TYPE DMC_Ins :
STRUCT
	DMC_Inputs : DriveInputs;
	DMC_POS_Status : PositionStatus;
	DMC_Drv_Status : DriveStatus;
END_STRUCT
END_TYPE

(* stored: Version 1.1.0.1, ProductVersion 3.1.4024.9
   DUT DMC_Ins: Id {4bbc7a0f-705c-40cf-a9c2-df6e3b8d5498} *)
